Fanuc KAREL source: ka00002.KL

-- PROVISIONAL review KL for V1013-1; original PC SHA256 9dedbaf215c138fa54e2af098022f2b1d3fedf89d368b4381a1f42d1f9248e12
-- Incomplete behavior may be omitted. Consult companion uncertainty JSON. Do not deploy.
PROGRAM KA00002
%NOLOCKGROUP
VAR
  SRC : INTEGER
  DST : REAL
BEGIN
  -- UNRESOLVED_PC offsets 5-16; opcodes 2E,23
  -- UNRESOLVED_PC offsets 21-34; opcodes 21,64,23
  -- UNRESOLVED_PC offsets 39-43; opcodes 7F
END KA00002
